(* PLC project Unnamed, Unknown Unnamed 1 *)
(* stored: creationDateTime 2024-09-30T20:56:11, modificationDateTime 2024-09-30T22:11:55 *)

PROGRAM pwm_test_program
  VAR
    PWM_CONTROLLER0 : PWM_CONTROLLER;
    START_PB : BOOL;
    Channel : SINT := 3;
    FREQ : REAL := 1.0;
    DUTY_CYCLE : REAL := 50.0;
  END_VAR
  VAR
    SERVO AT %QX0.1 : BOOL := 0;
    ANALOG_PWM AT %QW0 : UINT := 65535;
  END_VAR

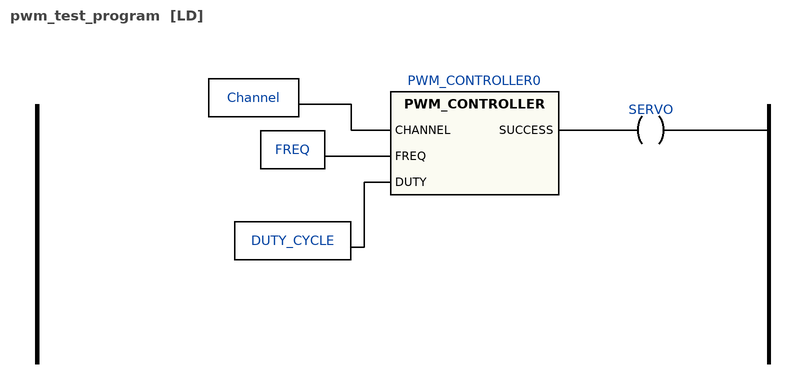
(* LD diagram, written out as Structured Text *)
PWM_CONTROLLER0(CHANNEL := Channel, FREQ := FREQ, DUTY := DUTY_CYCLE);
SERVO := PWM_CONTROLLER0.SUCCESS;
END_PROGRAM

CONFIGURATION Config0
  RESOURCE Res0 ON PLC
    TASK task0(INTERVAL := T#20ms, PRIORITY := 0);
    PROGRAM instance0 WITH task0 : pwm_test_program;
  END_RESOURCE
END_CONFIGURATION
